DATA_BLOCK "DB_BatchManager"
{ S7_Optimized_Access := 'TRUE' }
VERSION : 0.1
NON_RETAIN
"FB_BatchManager"

BEGIN

END_DATA_BLOCK

